{attribute 'GeneratedUsingTerminal: EL3751-0000-0020'}
{attribute addProperty BoxType "EL3751-0000-0020"}
{attribute addProperty Id "EtcSlaveTerminalBasePAI_StatusAT %I*PAI_Status_AE4AC1047PAI_Samples_1AT %I*PAI_Samples_EEA517254PAI_TimestampAT %I*PAI_Timestamp_6DC4D2968WcStateAT %I*WcState_9091E0EB2InfoDataAT %I*InfoData_BEF6B88E18"}
{attribute addProperty CRC "3945097629"}
{attribute addProperty Size "39"}
TYPE EL3751_EB25699D EXTENDS EtcSlaveTerminalBase :
STRUCT
	{attribute addProperty Name "PAI_Status"}
	PAI_Status : PAI_Status_AE4AC104;
	{attribute addProperty Name "PAI_Samples_1"}
	PAI_Samples_1 : PAI_Samples_EEA51725;
	{attribute addProperty Name "PAI_Timestamp"}
	PAI_Timestamp : PAI_Timestamp_6DC4D296;
	{attribute addProperty Name "WcState"}
	WcState : WcState_9091E0EB;
	{attribute addProperty Name "InfoData"}
	InfoData : InfoData_BEF6B88E;
END_STRUCT
END_TYPE

(* stored: Version 1.2.0.0, ProductVersion 3.1.4024.9
   DUT EL3751_EB25699D: Id {6375cac0-6864-4554-877f-8a610135c053} *)
